FUNCTION_BLOCK FB_CreateTepletate1 EXTENDS FB_Base IMPLEMENTS ITF_BaseCreateTemplateOfRecipe
VAR
END_VAR

METHOD CreateTamplateOfRecipe : BOOL
VAR_INPUT
	itfRecipe				: ITF_BaseCreatingTemplateMethod;	//interfejs do obsługi receptur
END_VAR
VAR
	sttmpSkladnik			: ST_BaseDescriptor;
	uiNumberOfTeplates		: UINT;
END_VAR
//	utworzenie szablonu z podaną nazwą
THIS^.SetText (eLocation := E_BaseLocation.pl, wsDescription := "Nazwa szablonu PL");
THIS^.SetText (eLocation := E_BaseLocation.en, wsDescription := "Nazwa szablonu EN");
THIS^.SetText (eLocation := E_BaseLocation.de, wsDescription := "Nazwa szablonu DE");
itfRecipe.AddTemplate (stTexts	:= GVL.fbRecipe.GetTexts ());
uiNumberOfTeplates	:= itfRecipe.GetNumberOfTemplate ();

THIS^.SetTextIn (stIN := sttmpSkladnik, eLocation := E_BaseLocation.pl, wsDescription := "Nazwa skladnika 1 PL");
THIS^.SetTextIn (stIN := sttmpSkladnik, eLocation := E_BaseLocation.en, wsDescription := "Nazwa skladnika 1 EN");
THIS^.SetTextIn (stIN := sttmpSkladnik, eLocation := E_BaseLocation.de, wsDescription := "Nazwa skladnika 1 DE");
THIS^.SetMaxIn (stIN := sttmpSkladnik, rMax := 10000);
THIS^.SetMinIn (stIN := sttmpSkladnik, rMin := 1);
THIS^.SetValueIn (stIN := sttmpSkladnik, rValue := 1111);
THIS^.SetDefaultValueIn (stIN := sttmpSkladnik, rDefaultValue := 1111);
THIS^.SetUnitIn (stIN := sttmpSkladnik, sUnit := 'mm');
itfRecipe.AddIngredientToTemplate (uiNumber := uiNumberOfTeplates, stIngredient := sttmpSkladnik);

THIS^.SetTextIn (stIN := sttmpSkladnik, eLocation := E_BaseLocation.pl, wsDescription := "Nazwa skladnika 2 PL");
THIS^.SetTextIn (stIN := sttmpSkladnik, eLocation := E_BaseLocation.en, wsDescription := "Nazwa skladnika 2 EN");
THIS^.SetTextIn (stIN := sttmpSkladnik, eLocation := E_BaseLocation.de, wsDescription := "Nazwa skladnika 2 DE");
THIS^.SetMaxIn (stIN := sttmpSkladnik, rMax := 10000);
THIS^.SetMinIn (stIN := sttmpSkladnik, rMin := 1);
THIS^.SetValueIn (stIN := sttmpSkladnik, rValue := 1112);
THIS^.SetDefaultValueIn (stIN := sttmpSkladnik, rDefaultValue := 1112);
THIS^.SetUnitIn (stIN := sttmpSkladnik, sUnit := 'mm/s');
itfRecipe.AddIngredientToTemplate (uiNumber := uiNumberOfTeplates, stIngredient := sttmpSkladnik);

THIS^.SetTextIn (stIN := sttmpSkladnik, eLocation := E_BaseLocation.pl, wsDescription := "Nazwa skladnika 3 PL");
THIS^.SetTextIn (stIN := sttmpSkladnik, eLocation := E_BaseLocation.en, wsDescription := "Nazwa skladnika 3 EN");
THIS^.SetTextIn (stIN := sttmpSkladnik, eLocation := E_BaseLocation.de, wsDescription := "Nazwa skladnika 3 DE");
THIS^.SetMaxIn (stIN := sttmpSkladnik, rMax := 10000);
THIS^.SetMinIn (stIN := sttmpSkladnik, rMin := 1);
THIS^.SetValueIn (stIN := sttmpSkladnik, rValue := 1113);
THIS^.SetDefaultValueIn (stIN := sttmpSkladnik, rDefaultValue := 1113);
THIS^.SetUnitIn (stIN := sttmpSkladnik, sUnit := 'ms');
itfRecipe.AddIngredientToTemplate (uiNumber := uiNumberOfTeplates, stIngredient := sttmpSkladnik);
END_METHOD

END_FUNCTION_BLOCK

(* stored: Version 1.1.0.1, ProductVersion 3.1.4024.15
   POU FB_CreateTepletate1: Id {a9f3d022-9d6a-4ed0-884e-e870ec758b64}, SpecialFunc None
   Method CreateTamplateOfRecipe: Id {d1dbda99-0797-426b-b2af-03ec540134dc} *)
